// TIA Portal V18 export
// export: Created 2026-06-03T07:11:55.5310194Z, ExportSetting WithDefaults, DisplayName Totally Integrated Automation Portal, DisplayVersion V18, DisplayName TIA Portal Openness, DisplayVersion V18, DisplayName TIA Portal Version Control Interface, DisplayVersion V18, DisplayName STEP 7 Professional, DisplayVersion V18, DisplayName STEP 7 Safety, DisplayVersion V18, DisplayName WinCC Professional, DisplayVersion V18
Screen "Test_Import_Screen"  800x600, Number=999
  ScreenLayer 
    GraphicView "Graphic view_1" at 0,0 size 800x600  Picture=Màn Tổng Quan Quy Trình_1
    Button "Button_2" at 153,529 size 107x46  Mode=Text, TextOff="VẬN HÀNH", TextOn="Text"
      on Click: ActivateScreen(Screen name := 02_Van_Hanh, Object number := 0)
    Button "Button_3" at 281,529 size 107x46  Mode=Text, TextOff="PID MỨC", TextOn="Text"
      on Click: ActivateScreen(Screen name := 03_PID_Muc_Nuoc, Object number := 0)
    Button "Button_6" at 409,528 size 107x46  Mode=Text, TextOff="TREND", TextOn="Text"
      on Click: ActivateScreen(Screen name := 04_Trend, Object number := 0)
    Button "Button_5" at 537,528 size 107x46  Mode=Text, TextOff="CẢNH BÁO", TextOn="Text"
      on Click: ActivateScreen(Screen name := 05_Canh_Bao_IO, Object number := 0)
    Circle "Circle_1" at 759,3 size 39x39
      RangeAppearanceAnimation "RangeAppearanceAnimation"
        tag bCheDoMoPhong
        0..0: back #d9d9d9, fore #181c31
        1..1: back #0000ff, fore #181c31
    Circle "Circle_2" at 718,3 size 39x39
      RangeAppearanceAnimation "RangeAppearanceAnimation"
        tag Loi_He_Thong
        0..0: back #d9d9d9, fore #181c31
        1..1: back #ff0000, fore #181c31
    Circle "Circle_3" at 677,3 size 39x39
      RangeAppearanceAnimation "RangeAppearanceAnimation"
        tag bSystemRun
        0..0: back #d9d9d9, fore #181c31
        1..1: back #00ff00, fore #181c31
    TextField "Text field_5" at 80,72 size 107x22  Text="Trạng Thái Mẻ"
    SymbolicIOField "Symbolic I/O field_1" at 43,107 size 197x36  CountVisibleItems=3, Mode=Output, OnValue=1, TextList=TL_Main_State, TextOff="0", TextOn="1"
      ProcessValue := Main_State
    IOField "I/O field_1" at 121,430 size 49x24  DataFormat=Decimal, FormatPattern=99.9, Mode=Output
      ProcessValue := Nhiet_Do_PV
    IOField "I/O field_2" at 121,456 size 49x24  DataFormat=Decimal, FormatPattern=99.9, Mode=Output
      ProcessValue := Ap_Suat_PV
    Circle "Circle_4" at 200,429 size 24x24
      RangeAppearanceAnimation "RangeAppearanceAnimation"
        tag Canh_Bao_Nhiet_Cao
        0..0: back #d9d9d9, fore #181c31
        1..1: back #ffff00, fore #181c31
    Circle "Circle_5" at 200,457 size 24x24
      RangeAppearanceAnimation "RangeAppearanceAnimation"
        tag Canh_Bao_Ap_Cao
        0..0: back #d9d9d9, fore #181c31
        1..1: back #ffff00, fore #181c31
    Rectangle "Rectangle_1" at 248,415 size 283x91
    TextField "Text field_8" at 374,416 size 39x20  Text="STEP"
    Rectangle "Rectangle_2" at 266,464 size 33x34
      RangeAppearanceAnimation "RangeAppearanceAnimation"
        tag Step0_IDLE
        0..0: back #d9d9d9, fore #181c31
        1..1: back #00ff00, fore #181c31
    Rectangle "Rectangle_3" at 318,464 size 33x34
      RangeAppearanceAnimation "RangeAppearanceAnimation"
        tag Step1_Thuc
        0..0: back #d9d9d9, fore #181c31
        1..1: back #00ff00, fore #181c31
    Rectangle "Rectangle_4" at 373,464 size 33x34
      RangeAppearanceAnimation "RangeAppearanceAnimation"
        tag Step2_Giu
        0..0: back #d9d9d9, fore #181c31
        1..1: back #00ff00, fore #181c31
    Rectangle "Rectangle_5" at 429,464 size 33x34
      RangeAppearanceAnimation "RangeAppearanceAnimation"
        tag Step3_KetThuc
        0..0: back #d9d9d9, fore #181c31
        1..1: back #00ff00, fore #181c31
    Rectangle "Rectangle_6" at 482,464 size 33x34
      RangeAppearanceAnimation "RangeAppearanceAnimation"
        tag StepErr_Loi
        0..0: back #d9d9d9, fore #181c31
        1..1: back #ff0000, fore #181c31
    TextField "Text field_9" at 266,446 size 28x16  Text="IDLE"
    TextField "Text field_10" at 307,445 size 50x16  Text="Gia Nhiệt"
    TextField "Text field_11" at 360,445 size 56x16  Text="Chưng Cất"
    TextField "Text field_12" at 421,445 size 47x16  Text="Kết Thúc"
    TextField "Text field_13" at 487,445 size 20x16  Text="Lỗi"
    Rectangle "Rectangle_7" at 676,345 size 120x121
    TextField "Text field_14" at 682,346 size 103x22  Text="Mức nước PV"
    IOField "I/O field_3" at 708,365 size 59x19  DataFormat=Decimal, FormatPattern=9.9, Mode=Output
      ProcessValue := Muc_Nuoc_PV
    TextField "Text field_15" at 682,381 size 106x22  Text="Mức Nước SP"
    IOField "I/O field_4" at 708,400 size 60x22  DataFormat=Decimal, FormatPattern=9.9, Mode=Output
      ProcessValue := Muc_Nuoc_SP
    TextField "Text field_16" at 707,419 size 56x22  Text="Van Xả"
    IOField "I/O field_5" at 707,439 size 60x22  DataFormat=Decimal, FormatPattern=99.9, Mode=Output
      ProcessValue := Van_Xa_OP
    TextField "Text field_17" at 744,399 size 17x22  Text="m"
    TextField "Text field_18" at 744,362 size 17x22  Text="m"
    TextField "Text field_19" at 748,439 size 18x22  Text="%"
    TextField "Text field_20" at 164,457 size 31x22  Text="Bar"
    TextField "Text field_21" at 166,431 size 23x22  Text="°C"
    Bar "Bar_1" at 561,324 size 59x107  CountSubDivisions=1, IntegerDigits=2, LargeTickLabelingStep=1, MaximumValue=0.5, Precision=1
      ProcessValue := Muc_Nuoc_PV
    GraphicIOField "Graphic I/O field_2" at 698,236 size 90x80  Mode=Output, OnValue=1, PictureList=GL_Bom_Lam_Mat
      RangeAppearanceAnimation "RangeAppearanceAnimation"
        tag 
      ProcessValue := Bom_Lam_Mat_M
    TextField "Text field_1" at 194,3 size 375x30  Text="HỆ THỐNG CHƯNG CẤT TINH DẦU"
    TextField "Text field_2" at 679,42 size 34x22  Text="Run"
    TextField "Text field_3" at 717,42 size 40x22  Text="Fault"
    TextField "Text field_4" at 760,42 size 31x22  Text="Sim"
    TextField "Text field_6" at 52,431 size 73x22  Text="Nhiệt độ:"
    TextField "Text field_7" at 59,456 size 65x22  Text="Áp suất:"
    GraphicIOField "Graphic I/O field_3" at 4,248 size 227x174  Mode=Output, OnValue=1, PictureList=GL_Noi_Hoi
      ProcessValue := HMI_Boiler_GFX
    Rectangle "Rectangle_8" at 23,526 size 114x52
    GraphicIOField "Graphic I/O field_1" at 220,326 size 44x38  Mode=Output, OnValue=1, PictureList=GL_Van_Hoi
      ProcessValue := HMI_SteamValve_GFX
    GraphicIOField "Graphic I/O field_4" at 295,122 size 208x294  Mode=Output, OnValue=1, PictureList=GL_Bon_Trung_Cat
      ProcessValue := HMI_DistillTank_GFX
    GraphicIOField "Graphic I/O field_5" at 490,78 size 238x160  Mode=Output, OnValue=1, PictureList=GL_Bon_Ngung_Tu
      ProcessValue := HMI_Condenser_GFX
    GraphicIOField "Graphic I/O field_6" at 697,235 size 91x81  Mode=InOutput, OnValue=1, PictureList=GL_Bom_Lam_Mat
      ProcessValue := HMI_CoolingPump_GFX
    GraphicIOField "Graphic I/O field_7" at 636,400 size 48x29  Mode=InOutput, OnValue=1, PictureList=GL_Van_Xa
      ProcessValue := HMI_DrainValve_GFX
    GraphicIOField "Graphic I/O field_8" at 1,-1 size 54x43  Mode=Output, OnValue=1, PictureList=GL_Alarm
      ProcessValue := HMI_Alarm_GFX
    Button "Button_1" at 27,529 size 107x46  Mode=Text, TextOff="TỔNG QUAN", TextOn="Text"
      on Click: ActivateScreen(Screen name := , Object number := 0)
    Button "Button_4" at 732,552 size 65x30  Mode=Text, TextOff="EXIT", TextOn="Text"
      on Click: StopRuntime(Mode := 0)
  SoftKey "Softkey_F9"  KeyCode=204
